// TIA Portal V15.1 export
// export: Created 2025-12-09T12:23:25.2728467Z, ExportSetting WithDefaults, WithReadOnly, DisplayName Totally Integrated Automation Portal, DisplayVersion V15.1, DisplayName TIA Portal Openness, DisplayVersion V15.1, DisplayName SINAMICS Startdrive Advanced, DisplayVersion V15.1, DisplayName SINAMICS DCC, DisplayVersion V15.1, DisplayName G130, G150, S120, S150, SINAMICS MV, S210, DisplayVersion V15.1, DisplayName G110M, G120, G120C, G120D, G120P, DisplayVersion V15.1, DisplayName STEP 7 Professional, DisplayVersion V15.1, DisplayName STEP 7 Safety, DisplayVersion V15.1, DisplayName WinCC Professional, DisplayVersion V15.1, DisplayName SIMATIC Visualization Architect, DisplayVersion V15.1
DATA_BLOCK "[nome_robo]_[numero_fm]#FB_Status_Global_DB"   // DB[numero_db]
{ S7_Optimized_Access := 'TRUE' }
AUTHOR : VASS_V05
FAMILY : STATUSGL
VERSION : 0.0
// Gesamt
// stored: AutoNumber false, CodeModifiedDate 2018-05-04T14:48:36.8234611Z, CompileDate 2019-04-01T14:36:11.4315261Z, CreationDate 2017-04-11T19:23:05.038059Z, DBAccessibleFromOPCUA true, DownloadWithoutReinit false, InstanceOfName FB_Status_Global, InstanceOfNumber 126, InstanceOfType FB, InterfaceModifiedDate 2018-05-04T14:42:01.5818586Z, IsConsistent true, IsKnowHowProtected false, IsRetainMemResEnabled false, MemoryReserve 0, ModifiedDate 2018-05-04T14:48:36.8234611Z, ParameterModified 2018-05-04T14:42:01.5818586Z, StructureModified 2018-05-04T14:42:01.5818586Z, UDAEnableTagReadback false
"FB_Status_Global"
   // VAR_INPUT
   //    Frg { ExternalAccessible := 'False'; ExternalVisible := 'False'; ExternalWritable := 'False'} : Bool;
   //    Cfg { ExternalAccessible := 'False'; ExternalVisible := 'False'; ExternalWritable := 'False'} : Word;
   // END_VAR
   // VAR_IN_OUT
   //    Status { ExternalAccessible := 'False'; ExternalVisible := 'False'; ExternalWritable := 'False'} : Bool;
   // END_VAR
   // VAR RETAIN
   //    "HMI-UDT" : "HMI-UDT_Status_Global";
   //    xHM_Tastendruck { ExternalAccessible := 'False'; ExternalVisible := 'False'; ExternalWritable := 'False'} : Bool;
   // END_VAR
   // VAR
   //    R_TRIG_SR { ExternalAccessible := 'False'; ExternalVisible := 'False'; ExternalWritable := 'False'} : "R_Trig";
   //    "255" { ExternalAccessible := 'False'; ExternalVisible := 'False'; ExternalWritable := 'False'} : Bool;
   // END_VAR
BEGIN
END_DATA_BLOCK
